// TwinCAT 3 PLC project Sewts_PLC
// ProgramVersion: 3.1.4023.0
// libraries:
//   Tc2_Standard, * (Beckhoff Automation GmbH)
//   Tc2_System, * (Beckhoff Automation GmbH)
//   Tc2_TcpIp, * (Beckhoff Automation GmbH)
//   Tc3_Module, * (Beckhoff Automation GmbH)
// project tree:
//   GVLs/ GVX.TcGVL, input.TcGVL, output.TcGVL
//   / PlcTask.TcTTO
//   POUs/ MAIN.TcPOU
//   TOOLS/TCP/ FB_TCP_COM.TcPOU
//   TOOLS/TCP/ST/ Sewts_TCP.TcGVL, strBufferHeader.TcDUT, strQueueContent.TcDUT, strQueueContentDetail.TcDUT (not stored), strQueueDetail.TcDUT, strQueueDetailExtended.TcDUT
// real-time tasks:
//   TASK PlcTask: cycle T#10ms, priority 20, ADS port 350

CONFIGURATION Sewts_PLC
    RESOURCE PLC ON TwinCAT3
        TASK PlcTask(INTERVAL := T#10ms, PRIORITY := 20);
        PROGRAM MAIN WITH PlcTask : MAIN;
    END_RESOURCE
END_CONFIGURATION

// ---- TOOLS/TCP/ST/strBufferHeader.TcDUT
TYPE strBufferHeader :
	STRUCT
		arbyDATA	: ARRAY[1..Sewts_TCP.MAX_BUFFER_SIZE] OF BYTE;
		bJob		: BOOL;		
	END_STRUCT
END_TYPE

// ---- TOOLS/TCP/ST/strQueueContent.TcDUT
	TYPE strQueueContent  :
	STRUCT
		uiCount		: UINT;
		uiMaxCount  : UINT;				(* information only, can be used to understand the queue load *)
		iTelHandle	: UDINT;			(* to maintain a unique msg handle 		*)
		iLastHAndle : UDINT; 			(* handle of last telegram fired 		*)
		STACK		: ARRAY  [0 .. Sewts_TCP.MAX_QUEUE_SIZE] OF strQueueContentDetail;
	END_STRUCT
END_TYPE

// ---- TOOLS/TCP/ST/strQueueDetail.TcDUT
TYPE strQueueDetail :
	STRUCT
		uiPrio			: UINT;				(* Option Sendepriorität 				*)
		uiMsgHandle 	: UDINT;			(* unique msg handle,  					*)
		pDATA			: POINTER TO BYTE ;	(* pointer on real data 				*)
		szDATA			: UDINT;			(* Length of data from pointer reference*)
	END_STRUCT
END_TYPE

// ---- TOOLS/TCP/ST/strQueueDetailExtended.TcDUT
TYPE strQueueDetailExtended EXTENDS strQueueDetail :
	STRUCT
		aDATA			: ARRAY [0..Sewts_TCP.MAX_QueueData] OF BYTE ;	(* Data *)
	END_STRUCT
END_TYPE

// ---- GVLs/GVX.TcGVL
{attribute 'qualified_only'}
VAR_GLOBAL
	arrbySend_Data			: ARRAY [0..Sewts_TCP.MAX_QUEUE_SIZE] OF BYTE;
	arrbyReceive_Data		: ARRAY [0..Sewts_TCP.MAX_QUEUE_SIZE] OF BYTE;
END_VAR

// ---- GVLs/input.TcGVL
{attribute 'qualified_only'}
VAR_GLOBAL
	bsSensor		: BOOL; //s sensor for detection cylinder NO
	bM2Spindisk		:BOOL; // spins disk Motor
	bM1Motor		:BOOL; // M1 motor 
	
END_VAR

// ---- GVLs/output.TcGVL
{attribute 'qualified_only'}
VAR_GLOBAL
	bM1Motor		:BOOL; // M2 motor 
	bM2Motor 		:BOOL;	//M2 Motor
END_VAR

// ---- TOOLS/TCP/ST/Sewts_TCP.TcGVL
VAR_GLOBAL CONSTANT 
	
	MAX_Bool_SIZE	:UINT := 31;	(* size of send & recceive buffer -> see "strBufferHeader.arbyDATA"  *)
		
END_VAR

// ---- POUs/MAIN.TcPOU


(*sewts Gmbh pick and plac project from Feed-rotating table*)
(*Author :Vaibhav Tank*)
PROGRAM MAIN
VAR
	TCP_COM 		:FB_TCP_COM;
	

	bEanable_Sever		:BOOL   := FALSE;
	uinPort				:UINT   :=9800;				
	sIP_Address			:STRING :='127.0.0.1';							
	bTCP_COM_Connected	:BOOL;
	bTCP_COM_Error		:BOOL;
	iTCP_COM_ErrId		:UDINT;
	stTCP_COM_sError	:STRING(80);
	
	(*timer*)
	Timer100ms           :TON;
	Timer500ms			 :TON;
	
	
	(*initialisation for the array in Global *)
	i 					: INT ;
		
END_VAR

TCP_COM(bEnable:= TRUE,
		nPort:=uinPort,
		sIPAddress:=sIP_Address,
		tFireDelay:=);
		
		(*Output from the function block TCP/IP communication*)
        bTCP_COM_Error		:=TCP_COM.bError;
        iTCP_COM_ErrId		:=TCP_COM.nErrId;
        stTCP_COM_sError	:=TCP_COM.sError;
		bTCP_COM_Connected 	:= TCP_COM.bConnected;
				
		(* Configuration of Timer100ms *)
Timer100ms(IN := TRUE, PT := T#100MS);
Timer500ms(IN := TRUE, PT := T#100MS);

IF Timer100ms.Q THEN
   TCP_COM.WriteInQueue_by_Pointer(pDATA:=ADR(GVX.arrbySend_Data),szDATA:=SIZEOF(GVX.arrbySend_Data),Prio:=1);
   TCP_COM.ptReceiveBuffer := ADR(GVX.arrbyReceive_Data);
	 Timer100ms(IN := FALSE);
	 
END_IF

IF Timer100ms.Q THEN
	 GVX.arrbySend_Data[0].0 := NOT  GVX.arrbySend_Data[0].0;
	 Timer500ms(IN := FALSE);
END_IF
TCP_COM.WriteInQueue_by_Pointer(pDATA:=ADR(GVX.arrbySend_Data),szDATA:=SIZEOF(GVX.arrbySend_Data),Prio:=1);

END_PROGRAM

// ---- TOOLS/TCP/FB_TCP_COM.TcPOU
// 18.4.2019    NetString lenght without endcharacters
// 3.4.2019     + Option "sNetStringSep"
// 26.3.2019   	+ Option "bAddNetStingLen"
//				+ Option "enuOptions.CheckAndTerminate_Custom"				
// 
// former known as fb_TCPIP_COMMUNICATION
FUNCTION_BLOCK FB_TCP_COM
VAR_INPUT
	
	bEnable			:BOOL		:= TRUE;	(* This function *)
	(* com parameter  *)
	bAsClient		:BOOL		:= FALSE;	(* FALSE -> TCP - Server / TCP-Client *)	
	nPort			:UINT		:= 2000;		(* SERVER: port to provide / CLIENT: port on server  				*)
	sIPAddress		:STRING (80):= '127.0.0.1';	(* SERVER: own network address to use / CLIENT: address of server 	*)
	(* send options*)
	tFireDelay		:TIME		:= T#0S;	(* betwenn two messages *)
	bCompactMessage	:BOOL		:= TRUE;	(* forces to send all messages AS one telegram - partner has to splitt messages!!!  *)
	xEOT			:BYTE		:= 16#03;	(* end of text character, use option "enuOptions.CheckAndTerminate_X" to activate	*)
	bAddNetStingLen	:BOOL		:= FALSE;	(* adds string len XX:yyyyyy in front of transmission								*)
	sNetStringSep	:STRING(1)	:= ':';
	ptReceiveBuffer	:POINTER TO strBufferHeader;	(* find receive data and coordination flag in here  *)
END_VAR

VAR_OUTPUT
	bConnected		:BOOL;
	bError			:BOOL;	
	nErrId			:UDINT;				(* FB_SocketConnect Error ID  		                                         *)
	sError			:STRING[80];		(* Error text (out of TC help system 	                                     *)
END_VAR
VAR
	// TCP Connection
	//tcp_ClientConnection	:FB_ClientServerConnection;
	
	// https://infosys.beckhoff.com/index.php?content=../content/1031/tf6310_tc3_tcpip/27021597848412555.html&id=
	(* client *)
	fbConnect       	: FB_SocketConnect 	:= ( sSrvNetId := '' );
   	fbClose        		: ARRAY[1..2] OF  FB_SocketClose;
	(* server *)
	fbListen			: FB_SocketListen;
	fbAccept			: FB_SocketAccept;
    fbSocketSend 		: FB_SocketSend 	:= ( sSrvNetID := '', tTimeout := DEFAULT_ADS_TIMEOUT );
    fbSocketReceive 	: FB_SocketReceive 	:= ( sSrvNetID := '', tTimeout := DEFAULT_ADS_TIMEOUT );
	fbSocketCloseAll : FB_SocketCloseAll;
	
	hListener          	: T_HSOCKET;
	hSocket         	: T_HSOCKET;
	
	x:int; (* xxx *)

	
	
	//Helpers
	iSTEP				:INT	:= 3;	(* main sequence*)
	ioldStep			:INT;
	tSTEP				:TON;
	TimeInStep 			:TIME;	
	i,uiLEN				:UINT; 
	strDiagnose			:STRING; 
	udiSLEN 			:UDINT; (* num of bytes to befired *)
	udiHelp				:UDINT; 
	aServiceBuffer  	:ARRAY[0..Sewts_TCP.MAX_QueueData] OF BYTE ;	(* DATA for queue entry*)
	
	//Data Structures
	strSendQueue		:strQueueContent;
	strSendBuffer		:strBufferHeader;

	nPort_OLD			:UINT;				
	sIPAddress_OLD		:STRING;	
	bAsClient_OLD		:BOOL;

	sNetString			:STRING(10)	:= '';
	iTerminaterNetLen	:UDINT;

	sSrvNetId			:STRING		:= ''; 	
END_VAR

VAR CONSTANT 
	STEP_Error 		:INT 	:= -2;	
	STEP_ONConnect	:INT	:= 10;
	STEP_Disconnect	:INT	:= 21;		
	STEP_WAIT_SEND	:INT   	:= 11; 
	TimeOut			:TIME	:= T#2S;
	tClientLookup	:TIME 	:= T#5100MS; (* (server)  timeout to enable accept   *)
END_VAR

TimingSystem();

CheckReceiveData();

CASE iSTEP OF
	-3:	(*******************************************************)
	 	fbSocketCloseAll( sSrvNetId:= '', bExecute:= TRUE, tTimeout:= T#10S );
		IF NOT fbSocketCloseAll.bBusy THEN
			iSTEP	:= iSTEP+1;
		END_IF;		

	STEP_Error: (** -2 *****************************************************)	 
	 	strDiagnose := 'STEP ERROR ';
		fbSocketCloseAll( bExecute:= FALSE );
		FOR i := 1  TO 2 DO 
			fbClose[i].sSrvNetId 	:= sSrvNetId;
			fbClose[i].tTimeout		:= DEFAULT_ADS_TIMEOUT;
			fbClose[i]( bExecute	:= FALSE );
			
			CASE i OF 
				1: fbClose[i].hSocket:= hListener;
				2: fbClose[i].hSocket:= hSocket;
			END_CASE
			fbClose[i]( bExecute	:= TRUE);
		END_FOR; 	
		(* reset all executes *)
		fbConnect		(bExecute 	:= FALSE);
		
		iSTEP := iSTEP + 1; 
		
	-1: (*******************************************************)
		strDiagnose := 'error pause';
		FOR i := 1  TO 2 DO 
			fbClose[i]( bExecute	:= FALSE );
		END_FOR; 
		bConnected	:= FALSE;
		
		IF TimeInStep > TimeOut THEN
			bError	:= FALSE;
			iSTEP 	:= 0;
		END_IF

	0: 	(*******************************************************)
		strDiagnose := 'wait for enable';
		IF bEnable THEN
			iSTEP := iSTEP + 1; 
		END_IF
		
	1: 	(*******************************************************)
		strDiagnose := 'start / init';

		nPort_OLD			:= nPort;				
		sIPAddress_OLD		:= sIPAddress;	
		bAsClient_OLD		:= bAsClient;	
 		bConnected			:= FALSE;
		
		IF bAsClient THEN 
			iSTEP := iSTEP+1;
		ELSE
			iSTEP := 4;	
		END_IF; 		
		
	2: 	(*******************************************************)
		strDiagnose := 'Connect as CLIENT to a SERVER';
		fbConnect ( bExecute 	:= FALSE );
		fbConnect (	bExecute	:= TRUE,
					sSrvNetId	:= sSrvNetId,
					sRemoteHost	:= sIPAddress,
					nRemotePort	:= nPort);
	
		iSTEP	:= iSTEP + 1; 

	3: 	(*******************************************************)
		strDiagnose := 'Connect as CLIENT end';
		fbConnect ( bExecute 	:= FALSE );
       	IF NOT fbConnect.bBusy THEN
            IF NOT fbConnect.bError THEN
                bConnected 	:= TRUE;
                hSocket    	:= fbConnect.hSocket;
				iSTEP		:= STEP_ONConnect;	(* >> OnConnect >> *)
            ELSIF TimeInStep	> TimeOut THEN
				iSTEP		:=  STEP_Error; (* ReLoop *)
           END_IF
         END_IF;
	
	4: (*******************************************************)
		strDiagnose := 'Provide a SERVER';
	   (*******************************************************)
		fbAccept (bExecute		:= FALSE);
		fbListen (bExecute 		:= FALSE);

		fbListen (sSrvNetId		:= sSrvNetId,
					sLocalHost	:= sIPAddress,
					nLocalPort	:= nPort,
					tTimeout   	:= t#30s,
					bExecute	:= TRUE );
					
		iSTEP := iSTEP+1;
	5: (*******************************************************)
		strDiagnose := 'Wait for listener';
			fbListen(  bExecute := FALSE  );
			IF NOT fbListen.bBusy THEN
				IF NOT fbListen.bError THEN
					hListener 	:= fbListen.hListener;
					iStep 		:= iSTEP + 1;
				ELSE
					(*---------------------------------------------*)
					(* Report error to the outsiede                *)
					(*---------------------------------------------*)
					nErrId := fbListen.nErrId;
					IF nErrId = 16#8003 THEN //Port is already occupied 
						iSTEP:= -3;
					ELSE
						iStep := -1;
					END_IF;
				END_IF
			END_IF

	6:	(*******************************************************) 
		strDiagnose	:= 'enable acceptance of clients';
		fbAccept (bExecute		:= FALSE);
		fbAccept (hListener		:= hListener,
					 bExecute	:= TRUE ,
					tTIMEout	:= T#5S	);
						
			iStep	:=	iSTEP+1;

	7: (* wait for client connection *)
			fbAccept (bExecute  := FALSE);

			IF NOT  fbAccept.bBusy THEN  
				IF fbAccept.bError THEN (*FB_SocketAccept returned error!*)
					iStep := -2;
				ELSIF fbAccept.bAccepted THEN 
					hSocket 	:= fbAccept.hSocket;
					iStep  		:= 10;
					RETURN;
				END_IF;

			END_IF;
			
			IF TimeInStep >= tClientLookup  THEN
		 	   iStep := 6 ; (* enable accept again *)
			END_IF;

		
	(*******************************************************)		
	10: (* (10 )STEP_ONConnect *)
		strDiagnose := 'OnConnectEvent';
		bconnected 	:=TRUE;

		OnConnectEvent();
		iSTEP 		:= iSTEP+1; 

	11: (*******************************************************)	
		strDiagnose := 'Check Queue for data to send ';
		IF strSendQueue.uiCount > 0 THEN
			OnGetNextEvent();		// quicksort
			PrepareSendBuffer();	
	
			fbSocketSend( bExecute 	:= FALSE );
			fbSocketSend( hSocket 	:= hSocket,
						  pSrc 		:= ADR(strSendBuffer.arbyDATA),
						  cbLen 	:= udiSLEN,
						bExecute	:= TRUE );
						
			iSTEP	:= iSTEP + 1;
		END_IF;
		
	12: (*******************************************************)
      	fbSocketSend( bExecute 	:= FALSE );
		
   		IF NOT fbSocketSend.bBusy THEN
            IF NOT fbSocketSend.bError THEN
				IF tFireDelay <= T#0S THEN 
					iSTEP 	:= STEP_WAIT_SEND; (* ReLoop *)
				ELSE
					iSTEP 	:= iSTEP+1; 
				END_IF;
            ELSE
				iSTEP	:= STEP_Error;
            END_IF
        END_IF
		
	13: strDiagnose := 'Fire delay....';
		IF  TimeInStep > tFireDelay THEN 
				iSTEP 	:= STEP_WAIT_SEND; (* ReLoop *)
		ELSIF CheckParameterChange() THEN 
				iSTEP  := STEP_Error;
		END_IF;
ELSE 
		iSTEP := STEP_ERROR; 
END_CASE

METHOD PRIVATE CheckOptions : UINT
VAR_INPUT
	Option		:enuOptions;		(* Support Optios: see declaration for more details  *)
END_VAR
VAR_IN_OUT
	xLEN		:UINT; 
END_VAR

VAR
	xSize		:uint; 
END_VAR
	CheckOptions	:= 0;
	xSize			:= SIZEOF(aServiceBuffer);

CASE Option OF
		(*NoAction----------------------------------------------------------------------------------------------------------------------*)
	enuOptions.NONE: ;
		(*CheckLenByNul----------------------------------------------------------------------------------------------------------------------*)
	enuOptions.CheckNull:
			FOR i := 1 TO xSize DO
				IF aServiceBuffer[i]   = 0 THEN
					xLEN := i ;
	
					EXIT;
				END_IF;
			END_FOR;
		(*CheckLenByCRLF-----------------------------------------------------------------------------------------------------------------------*)
	enuOptions.CheckCRLF:
			FOR i := 1 TO xSize DO
				IF aServiceBuffer[i]   = 13 AND
					aServiceBuffer[i+1] = 10 THEN
					xLEN := i +2;
					EXIT;
				END_IF;
			END_FOR;
		(*CheckLenTerminateCRLF------------------------------------------------------------------------------------------------------------------------*)
	enuOptions.CheckAndTerminate_CRLF:
		FOR i := 1 TO xSize DO
			IF aServiceBuffer[i]   = 0 THEN
			(* check if  *)
				IF aServiceBuffer[i-2] = 16#D AND aServiceBuffer[i-1] = 16#A THEN
					//xLEN := i-1 ;
					EXIT; //already added
				END_IF;
				aServiceBuffer[i]	:= 16#D;
				aServiceBuffer[i+1]	:= 16#A;
				xLEN := i + 2 ;
				EXIT;
			END_IF;
		END_FOR;

	enuOptions.CheckAndTerminate_ETX:
		FOR i := 1 TO xSize DO
			IF aServiceBuffer[i]   = 0 THEN
			(* check if already added *)
				IF aServiceBuffer[i-1] = 16#3 THEN
					xLEN := i ;
					EXIT;
				END_IF;

				aServiceBuffer[i]	:= 16#3;
				xLEN := i+1 ;
				EXIT;
			END_IF;
		END_FOR;

	enuOptions.CheckAndTerminate_Custom:
		FOR i := 1 TO xSize DO
			IF aServiceBuffer[i]   = 0 THEN
			(* check if already added *)
				IF aServiceBuffer[i-1] = xEOT THEN
					xLEN := i ;
					EXIT;
				END_IF;

				aServiceBuffer[i]	:= xEOT;
				xLEN := i+1 ;
				EXIT;
			END_IF;
		END_FOR;
		
	END_CASE;
END_METHOD

METHOD INTERNAL CheckParameterChange : bool
CheckParameterChange := 	nPort_OLD			<> nPort OR 				
								sIPAddress_OLD		<> sIPAddress OR	
								bAsClient_OLD		<> bAsClient OR 
								bEnable				<> TRUE;
END_METHOD

ACTION CheckReceiveData:
(*---------------------------------------------*)
(* CheckReceiveData                            *)
(*---------------------------------------------*)

	IF bconnected AND (NOT fbSocketReceive.bBusy) AND (NOT fbSocketReceive.bExecute) THEN
		fbSocketReceive.bExecute :=TRUE;
	END_IF;

	IF (NOT bconnected) OR (fbSocketReceive.bBusy) THEN
		fbSocketReceive.bExecute :=FALSE;
	END_IF;
	
	fbSocketReceive(
				sSrvNetId	:= sSrvNetId,
				hSocket		:= hSocket,
				cbLen  		:= SIZEOF 	(ptReceiveBuffer^.arbyDATA),
				pDest  		:= ADR		(ptReceiveBuffer^.arbyDATA),
				tTimeout	:= T#5s);

	(* OnReceiveEvent *)				
	IF fbSocketReceive.nRecBytes >0  THEN 
		ptReceiveBuffer^.bJob := TRUE;
	END_IF
		
	(* Connection fail detection !!! *)
	IF 	(
		(fbSocketReceive.nErrId  = 16#8004) 
	OR 	(nPort_OLD		<> nPort)
	OR 	(sIPAddress_OLD	<> sIPAddress)
		)
	AND bConnected 
	AND iSTEP < 20 THEN
		bConnected 	:= FALSE;
		iSTEP 		:= STEP_Disconnect;
	END_IF;
END_ACTION

ACTION OnConnectEvent:
strSendQueue.uiCount := 0;
MemSet(destAddr := ADR(strSendQueue.STACK), fillByte := 0, n := SIZEOF (strSendQueue.STACK));
END_ACTION

ACTION OnGetNextEvent:
	QueTools_SortPrio_ASC(x := strSendQueue );
END_ACTION

ACTION PrepareSendBuffer:
(*---------------------------------------------*)
(* Prepare Send Buffer                         *)
(*---------------------------------------------*)
	(* CLR send buffer befor loading data into it *)
	MemSet(destAddr := ADR (strSendBuffer.arbyDATA), fillByte := 0, n := SIZEOF (strSendBuffer.arbyDATA));
	
	udiSLEN := 0 ; 
	WHILE strSendQueue.uiCount > 0 DO  
		(* pull lowest queue element *)
		strSendQueue.actEntry     := strSendQueue.STACK[1];
		strSendQueue.iLastHAndle  := strSendQueue.actEntry.uiMsgHandle;
				
		(* copy data from source mem into Sendbuffer *)
		MEMCPY(destAddr  := ADR (strSendBuffer.arbyDATA)+ udiSLEN ,srcAddr :=ADR(strSendQueue.actEntry.aDATA), n := strSendQueue.actEntry.uiDATA );
		
		
		(*---------------------------------------------*)
		(* DECREMENT Stack                             *)
		(*---------------------------------------------*)
		strSendQueue.uiCount    := strSendQueue.uiCount - 1;
		FOR i := 1 TO Sewts_TCP.MAX_QUEUE_SIZE -1 DO
			strSendQueue.STACK[i] := strSendQueue.STACK[i+1];
		END_FOR;
		
		FOR i := 0 TO Sewts_TCP.MAX_QueueData DO strSendQueue.STACK[Sewts_TCP.MAX_QUEUE_SIZE].aDATA[i] := 0; END_FOR; 
		strSendQueue.STACK[Sewts_TCP.MAX_QUEUE_SIZE].byOption	:= 0;
		strSendQueue.STACK[Sewts_TCP.MAX_QUEUE_SIZE].uiPrio	:= 0;
		strSendQueue.STACK[Sewts_TCP.MAX_QUEUE_SIZE].uiDATA	:= 0;

		(*---------------------------------------------*)
		(* Lenght check *)
		(*---------------------------------------------*)
		IF ( strSendQueue.uiCount > 0	(* more entrys? *)
		AND  strSendQueue.STACK[1].uiDATA> 0 
		AND  strSendQueue.STACK[1].uiDATA + udiSLEN > Sewts_TCP.MAX_BUFFER_SIZE) 

		THEN 
			EXIT; 
		END_IF

		(*---------------------------------------------*)
		(* Paramater bCompactMessage                   *)
		(*---------------------------------------------*)
		IF NOT bCompactMessage THEN 
			EXIT; 
		END_IF
		
	END_WHILE;
END_ACTION

METHOD PRIVATE QueTools_SortPrio_ASC : BOOL
VAR_IN_OUT
	X			: strQueueContent;
END_VAR
VAR
	y			: strQueueContent;
	One			: strQueueContentDetail;
	LastCount	: UINT;
	bHandled	: ARRAY[1..Sewts_TCP.MAX_QUEUE_SIZE] OF BOOL;
	i			: UINT;
	j			: UINT;
	idx			: UINT;
END_VAR
QueTools_SortPrio_ASC :=FALSE;

	IF x.uiCount < 2 THEN
		RETURN ;
	END_IF;

	IF LastCount > x.uiCount THEN
		LastCount  := x.uiCount ;
	  	RETURN;
	END_IF;
		LastCount  := x.uiCount ;

	FOR i := 1 TO Sewts_TCP.MAX_QUEUE_SIZE DO
	  bHandled[i] := FALSE;
	END_FOR;

	y.uiCount := 0;
	J := 1;

	REPEAT

		IF NOT bHandled[J] THEN
			One := X.STACK[J];
			idx := J;

			FOR i := 1 TO x.uiCount DO
				IF (One.uiPrio > x.STACK[i].uiPrio) AND (NOT bHandled[i])  AND (j <> i)  THEN
					One  := x.STACK[i];
					idx  := i;
				END_IF;
			END_FOR;

			bHandled[idx] := TRUE;
			Y.uiCount := Y.uiCount +1;
			y.STACK[Y.uiCount] := One;
			J := 1;
		ELSE
			j := j + 1;
		END_IF;

	UNTIL y.uiCount = x.uiCount
	END_REPEAT;


	FOR i := 1 TO x.uiCount DO
		x.STACK[i] := y.STACK[i];
	END_FOR;

	QueTools_SortPrio_ASC := TRUE;
END_METHOD

ACTION TimingSystem:
	IF iSTEP <> ioldStep THEN
//			main.FileLogger.AddMessage(xChapter:= 'TCP STEP ',xMessage:= int_to_string(iSTEP));
			ioldStep := iSTEP ;
			tSTEP( IN := FALSE, PT := t#5s );
	END_IF;
	
	tSTEP( IN := TRUE, PT := T#60M );
	TimeInStep  := tSTEP.ET ;
END_ACTION

ACTION WaitForClient:
(*	
	tcp_server		(xEnable := TRUE, ipAddr 	:= sIPAddr, uiPort := nPort);
		tcp_connections	(xEnable := TRUE, hServer 	:= tcp_server.hServer);
	
		IF tcp_connections.xActive THEN
			hConnection 	:= tcp_connections.hConnection;
			bConnected		:= TRUE;
			iSTEP 			:= STEP_ONConnect;
			
		ELSIF tcp_connections.xError OR CheckParameterChange() THEN 
			iSTEP 			:= STEP_Error;

		END_IF;			
	
*)
END_ACTION

METHOD PUBLIC WriteInQueue_by_ByteArray : UDINT (* Message Handle *)
VAR_INPUT
	aDATA		: ARRAY[0..Sewts_TCP.MAX_QueueData] OF BYTE ;	(* DATA to be send *)
	uiDATA		: UINT;			    (* amout of byte to send, see also "Option" 		 *)
	Prio		: UINT ;	    	(* Optionale Parameter used for the quick sort       *)
END_VAR

VAR 
	uiLEN			:UINT;
END_VAR
	(* init *)
	WriteInQueue_by_ByteArray := 0;
	(* some basic checks *)
	IF strSendQueue.uiCount >= Sewts_TCP.MAX_QUEUE_SIZE THEN
   	   strSendQueue.uiCount := Sewts_TCP.MAX_QUEUE_SIZE ;
		RETURN;
	END_IF;

	IF  strSendQueue.uiCount < 0 THEN
		strSendQueue.uiCount := 0;
	END_IF;

	(* INC stack queue idx  *)
	strSendQueue.uiCount := strSendQueue.uiCount + 1 ;

	(* peak load detection*)
	IF 	strSendQueue.uiCount > strSendQueue.uiMaxCount THEN
		strSendQueue.uiMaxCount := strSendQueue.uiCount;
	END_IF ;

	(* unique handle *)
	strSendQueue.iTelHandle := strSendQueue.iTelHandle + 1;
	
	(*---------------------------------------------*)
	(* Data to internal buffer *)
	(*---------------------------------------------*)
	MemCpy(destAddr:=ADR(aServiceBuffer),srcAddr := ADR(aData),n:=SIZEOF(aData));
	uiLEN			:= uiDATA;
	

	(* fill stack element *)
	strSendQueue.STACK[strSendQueue.uiCount].uiPrio			:= Prio;
	strSendQueue.STACK[strSendQueue.uiCount].uiMsgHandle	:= strSendQueue.iTelHandle;
	strSendQueue.STACK[strSendQueue.uiCount].aDATA			:= aServiceBuffer ;				(* updated element *)
	strSendQueue.STACK[strSendQueue.uiCount].uiDATA			:= uiLEN;

	(* return handle *)
	WriteInQueue_by_ByteArray := strSendQueue.iTelHandle;
END_METHOD

METHOD PUBLIC WriteInQueue_by_Pointer : UDINT (* Message Handle *)
VAR_INPUT
	pDATA		: POINTER TO BYTE ;	(* Pointer to Data to be send *)
	szDATA		: UINT;				(* amout of byte to send, see also "Option" *)
	Prio		:UINT ;	    		(* Optionale Parameter used for the quick sort       *)
END_VAR

VAR 
	i			:UINT;
END_VAR

VAR CONSTANT
	MaxLength :UINT := 255; 
END_VAR
	(* init *)
	WriteInQueue_by_Pointer := 0;
	IF szData > MaxLength THEN 
		RETURN; 
	END_IF
	
	
	(* some basic checks *)
	IF strSendQueue.uiCount >= Sewts_TCP.MAX_QUEUE_SIZE THEN
   	   strSendQueue.uiCount := Sewts_TCP.MAX_QUEUE_SIZE ;
		RETURN;
	END_IF;

	IF  strSendQueue.uiCount < 0 THEN
		strSendQueue.uiCount := 0;
	END_IF;

	(* INC stack queue idx  *)
	strSendQueue.uiCount := strSendQueue.uiCount + 1 ;

	(* peak load detection*)
	IF 	strSendQueue.uiCount > strSendQueue.uiMaxCount THEN
		strSendQueue.uiMaxCount := strSendQueue.uiCount;
	END_IF ;

	(* unique handle *)
	strSendQueue.iTelHandle := strSendQueue.iTelHandle + 1;
	
	(*---------------------------------------------*)
	(* Data to internal buffer *)
	(*---------------------------------------------*)
	FOR i := 0 TO Sewts_TCP.MAX_QueueData DO  aServiceBuffer[i] :=0; END_FOR;
 	MemCpy(destAddr:= ADR(aServiceBuffer),srcAddr:= pDATA ,n := szDATA);
	uiLEN			:= szDATA;
	(*---------------------------------------------*)
	(* Supporting routines now in here!!!          *)
	(*---------------------------------------------*)
	CheckOptions( Option := Option, xLEN:=uiLEN);
	
	(*---------------------------------------------*)
	(* fill stack element                          *)
	(*---------------------------------------------*)	
	strSendQueue.STACK[strSendQueue.uiCount].uiPrio			:= Prio;
	strSendQueue.STACK[strSendQueue.uiCount].byOption 		:= Option;
	strSendQueue.STACK[strSendQueue.uiCount].uiMsgHandle	:= strSendQueue.iTelHandle;
	strSendQueue.STACK[strSendQueue.uiCount].aDATA			:= aServiceBuffer ;				(* updated element *)
	strSendQueue.STACK[strSendQueue.uiCount].uiDATA			:= uiLEN;

	(* return handle *)
	WriteInQueue_by_Pointer := strSendQueue.iTelHandle;
END_METHOD

METHOD PUBLIC WriteInQueue_by_String : UDINT (* Message Handle *)
VAR_INPUT
	sString		:STRING(255);		(* string to be send *)
	Prio		:UINT ;	    		(* Optionale Parameter used for the quick sort       *)
END_VAR

VAR 
	i			:UINT;
	
	
END_VAR
	(* init *)
	WriteInQueue_by_String := 0;
	(* some basic checks *)
	IF strSendQueue.uiCount >= Sewts_TCP.MAX_QUEUE_SIZE THEN
   	   strSendQueue.uiCount := Sewts_TCP.MAX_QUEUE_SIZE ;
		RETURN;
	END_IF;

	IF  strSendQueue.uiCount < 0 THEN
		strSendQueue.uiCount := 0;
	END_IF;

	(* INC stack queue idx  *)
	strSendQueue.uiCount := strSendQueue.uiCount + 1 ;

	(* peak load detection*)
	IF 	strSendQueue.uiCount > strSendQueue.uiMaxCount THEN
		strSendQueue.uiMaxCount := strSendQueue.uiCount;
	END_IF ;

	(* unique handle *)
	strSendQueue.iTelHandle := strSendQueue.iTelHandle + 1;
	
	(*---------------------------------------------*)
	(* Data to internal buffer *)
	(*---------------------------------------------*)
	FOR i := 0 TO Sewts_TCP.MAX_QueueData DO  aServiceBuffer[i] :=0; END_FOR;
 	MemCpy(destAddr:= ADR(aServiceBuffer),srcAddr:= ADR(sString),n :=  INT_TO_UINT (LEN(sString)));
	
	uiLEN			:= INT_TO_UINT(LEN(sString));
	(*---------------------------------------------*)
	(* Supporting routines now in here!!!          *)
	(*---------------------------------------------*)
	CheckOptions( Option := Option, xLEN:=uiLEN);
	
	(*---------------------------------------------*)
	(* fill stack element                          *)
	(*---------------------------------------------*)	
	strSendQueue.STACK[strSendQueue.uiCount].uiPrio			:= Prio;
	strSendQueue.STACK[strSendQueue.uiCount].byOption 		:= Option;
	strSendQueue.STACK[strSendQueue.uiCount].uiMsgHandle	:= strSendQueue.iTelHandle;
	strSendQueue.STACK[strSendQueue.uiCount].aDATA			:= aServiceBuffer ;				(* updated element *)
	strSendQueue.STACK[strSendQueue.uiCount].uiDATA			:= uiLEN;

	(* return handle *)
	WriteInQueue_by_String := strSendQueue.iTelHandle;
END_METHOD

END_FUNCTION_BLOCK
